PROGRAM MAIN
VAR
	i, j, x, y, sss : INT;
END_VAR

END_PROGRAM

(* stored: Version 1.1.0.1, ProductVersion 3.1.4022.16
   POU MAIN: Id {f569db27-f18a-4449-a510-316ce04bc5f8}, SpecialFunc None *)
